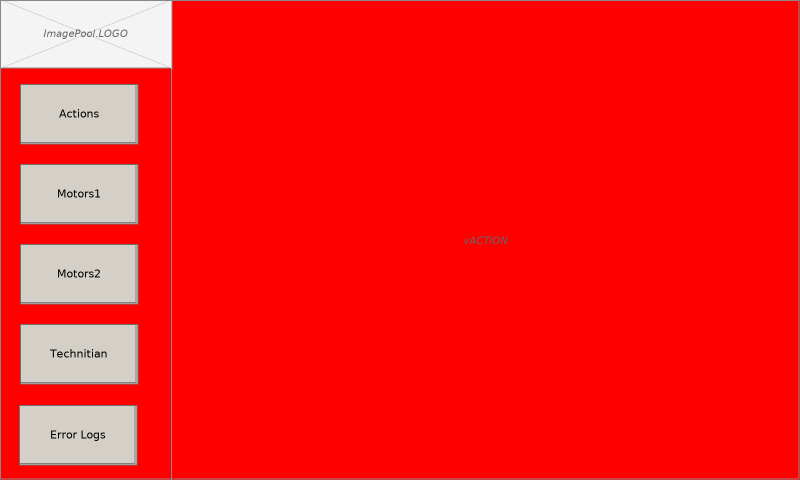
VISUALIZATION vCOMM  // 800x480
    Button (20,84 118x60), "Actions"
        OnMouseClick: FrameSelectionChange Selection=SelectedFrame=c79d80b7-c479-4a39-9ec5-d387b8e1dbac, GlobSel=AssignType=Directly, SelType=Locally
    Button (20,164 118x60), "Motors1", input disabled if: NOT ACTION1.bMANUAL
        OnMouseClick: FrameSelectionChange Selection=SelectedFrame=c79d80b7-c479-4a39-9ec5-d387b8e1dbac, Selection=1, GlobSel=AssignType=Directly, SelType=Locally
    Button (20,244 118x60), "Motors2", input disabled if: NOT ACTION2.bMANUAL
        OnMouseClick: FrameSelectionChange Selection=SelectedFrame=c79d80b7-c479-4a39-9ec5-d387b8e1dbac, Selection=2, GlobSel=AssignType=Directly, SelType=Locally
    Button (19,405 118x60), "Error Logs"
        OnMouseClick: FrameSelectionChange Selection=SelectedFrame=c79d80b7-c479-4a39-9ec5-d387b8e1dbac, Selection=3, GlobSel=AssignType=Directly, SelType=Locally
    Frame (171,-1 630x483)
        shows vACTION(vACTION := ACTION1, vACTION2 := ACTION2)
        shows vAXES1()
        shows vAXES2()
        shows vEVENT_LOGGER()
        shows vPISTONS()
    Button (20,324 118x60), "Technitian"
        OnMouseClick: FrameSelectionChange Selection=SelectedFrame=c79d80b7-c479-4a39-9ec5-d387b8e1dbac, Selection=4, GlobSel=AssignType=Directly, SelType=Locally
    Image (0,-1 172x69), image: ImagePool.LOGO
END_VISUALIZATION

(* stored: Version 1.1.0.1, ProductVersion 3.1.4024.12
   Visu vCOMM: Id {73f938e2-8269-424b-a9a0-181db6562291} *)
